# EPICS autosave request: iocBoot/iocRobot/auto_settings.req
file "robot.req", P=$(P), R=$(R)
file "robot_settings.req", P=$(P), R=$(R)
